{attribute 'c++_compatible'}
FUNCTION_BLOCK JsonSaxHandler_RobotState IMPLEMENTS ITcJsonSaxHandler
VAR_INPUT
END_VAR
VAR_OUTPUT
	parsedState :	STRING;
END_VAR
VAR
	bStateFound :			BOOL := FALSE;
	bCtrlexecstateFound :	BOOL := FALSE;
END_VAR

(* Example JSON

	{
		"_links": {
			"base": {
				"href": "http://127.0.0.1:80/rw/rapid/"
			},
			"self": {
				"href": "execution"
			}
		},
		"status": {
			"code": 294912
		},
		"state": [
			{
				"_type": "rap-execution",
				"_title": "execution",
				"ctrlexecstate": "stopped",
				"cycle": "forever"
			}
		]
	}

*)

{attribute 'TcTypeSystem'}
{attribute 'no-analysis'}
{attribute 'c++_compatible'}
{attribute 'minimal_input_size' := '4'}
{attribute 'pack_mode' := '4'}
{warning 'add method implementation '}
METHOD OnBool : HRESULT
VAR_INPUT
	value	: BOOL;
END_VAR
END_METHOD

{attribute 'TcTypeSystem'}
{attribute 'no-analysis'}
{attribute 'c++_compatible'}
{attribute 'minimal_input_size' := '4'}
{attribute 'pack_mode' := '4'}
{warning 'add method implementation '}
METHOD OnDint : HRESULT
VAR_INPUT
	value	: DINT;
END_VAR
END_METHOD

{attribute 'TcTypeSystem'}
{attribute 'no-analysis'}
{attribute 'c++_compatible'}
{attribute 'minimal_input_size' := '4'}
{attribute 'pack_mode' := '4'}
{warning 'add method implementation '}
METHOD OnEndArray : HRESULT
VAR_INPUT
	elementCount	: UDINT;
END_VAR
END_METHOD

{attribute 'TcTypeSystem'}
{attribute 'no-analysis'}
{attribute 'c++_compatible'}
{attribute 'minimal_input_size' := '4'}
{attribute 'pack_mode' := '4'}
{warning 'add method implementation '}
METHOD OnEndObject : HRESULT
VAR_INPUT
	memberCount	: UDINT;
END_VAR
END_METHOD

{attribute 'TcTypeSystem'}
{attribute 'no-analysis'}
{attribute 'c++_compatible'}
{attribute 'minimal_input_size' := '4'}
{attribute 'pack_mode' := '4'}
{warning 'add method implementation '}
METHOD OnKey : HRESULT
VAR_IN_OUT CONSTANT
	key	: STRING;
END_VAR
VAR_INPUT
	len	: UDINT;
END_VAR


IF (key = 'state') THEN
	bStateFound := TRUE;
END_IF

IF bStateFound AND (key = 'ctrlexecstate') THEN
	bCtrlexecstateFound := TRUE;
END_IF
END_METHOD

{attribute 'TcTypeSystem'}
{attribute 'no-analysis'}
{attribute 'c++_compatible'}
{attribute 'minimal_input_size' := '4'}
{attribute 'pack_mode' := '4'}
{warning 'add method implementation '}
METHOD OnLint : HRESULT
VAR_INPUT
	value	: LINT;
END_VAR
END_METHOD

{attribute 'TcTypeSystem'}
{attribute 'no-analysis'}
{attribute 'c++_compatible'}
{attribute 'minimal_input_size' := '4'}
{attribute 'pack_mode' := '4'}
{warning 'add method implementation '}
METHOD OnLreal : HRESULT
VAR_INPUT
	value	: LREAL;
END_VAR
END_METHOD

{attribute 'TcTypeSystem'}
{attribute 'no-analysis'}
{attribute 'c++_compatible'}
{attribute 'minimal_input_size' := '4'}
{attribute 'pack_mode' := '4'}
{warning 'add method implementation '}
METHOD OnNull : HRESULT
END_METHOD

{attribute 'TcTypeSystem'}
{attribute 'no-analysis'}
{attribute 'c++_compatible'}
{attribute 'minimal_input_size' := '4'}
{attribute 'pack_mode' := '4'}
{warning 'add method implementation '}
METHOD OnRawNumber : HRESULT
VAR_IN_OUT CONSTANT
	value	: STRING;
END_VAR
VAR_INPUT
	len	: UDINT;
END_VAR
END_METHOD

{attribute 'TcTypeSystem'}
{attribute 'no-analysis'}
{attribute 'c++_compatible'}
{attribute 'minimal_input_size' := '4'}
{attribute 'pack_mode' := '4'}
{warning 'add method implementation '}
METHOD OnStartArray : HRESULT
END_METHOD

{attribute 'TcTypeSystem'}
{attribute 'no-analysis'}
{attribute 'c++_compatible'}
{attribute 'minimal_input_size' := '4'}
{attribute 'pack_mode' := '4'}
{warning 'add method implementation '}
METHOD OnStartObject : HRESULT
END_METHOD

{attribute 'TcTypeSystem'}
{attribute 'no-analysis'}
{attribute 'c++_compatible'}
{attribute 'minimal_input_size' := '4'}
{attribute 'pack_mode' := '4'}
{warning 'add method implementation '}
METHOD OnString : HRESULT
VAR_IN_OUT CONSTANT
	value	: STRING;
END_VAR
VAR_INPUT
	len	: UDINT;
END_VAR

IF bCtrlexecstateFound THEN
	parsedState := value;
	OnString := S_FALSE;
END_IF
END_METHOD

{attribute 'TcTypeSystem'}
{attribute 'no-analysis'}
{attribute 'c++_compatible'}
{attribute 'minimal_input_size' := '4'}
{attribute 'pack_mode' := '4'}
{warning 'add method implementation '}
METHOD OnUdint : HRESULT
VAR_INPUT
	value	: UDINT;
END_VAR
END_METHOD

{attribute 'TcTypeSystem'}
{attribute 'no-analysis'}
{attribute 'c++_compatible'}
{attribute 'minimal_input_size' := '4'}
{attribute 'pack_mode' := '4'}
{warning 'add method implementation '}
METHOD OnUlint : HRESULT
VAR_INPUT
	value	: ULINT;
END_VAR
END_METHOD

METHOD Reset : bool
VAR_INPUT
END_VAR

VAR
	bStateFound: BOOL;
END_VAR

// Reset parsing state variables
bStateFound := FALSE;
bCtrlexecstateFound := FALSE;
END_METHOD

{attribute 'TcTypeSystem'}
{attribute 'no-analysis'}
{attribute 'c++_compatible'}
{attribute 'minimal_input_size' := '4'}
{attribute 'pack_mode' := '4'}
{warning 'add method implementation '}
METHOD TcAddRef : UDINT
END_METHOD

{attribute 'TcTypeSystem'}
{attribute 'no-analysis'}
{attribute 'c++_compatible'}
{attribute 'minimal_input_size' := '4'}
{attribute 'pack_mode' := '4'}
{warning 'add method implementation '}
METHOD TcQueryInterface : HRESULT
VAR_INPUT
	iid	: REFERENCE TO IID;
	pipItf	: POINTER TO PVOID;
END_VAR
END_METHOD

{attribute 'TcTypeSystem'}
{attribute 'no-analysis'}
{attribute 'c++_compatible'}
{attribute 'minimal_input_size' := '4'}
{attribute 'pack_mode' := '4'}
{warning 'add method implementation '}
METHOD TcRelease : UDINT
END_METHOD

END_FUNCTION_BLOCK

(* stored: Version 1.1.0.1, ProductVersion 3.1.4024.12
   POU JsonSaxHandler_RobotState: Id {b78b5962-e88f-45fd-9428-34c0448eb750}, SpecialFunc None
   Method OnBool: Id {a8bc2ecd-7eea-4493-a462-cbe13f3242fd}
   Method OnDint: Id {29d2b2b9-7237-49cd-9084-3f0f44c317b4}
   Method OnEndArray: Id {0391a5fd-ef8a-4caf-b3c9-24c17e026c2a}
   Method OnEndObject: Id {1c08a774-1c52-4db3-a402-0aa746cc3c2c}
   Method OnKey: Id {f813b109-3a0c-4827-a2f7-a3de3156088b}
   Method OnLint: Id {c93d24da-b0b2-4c38-b080-f3f010bd8a4c}
   Method OnLreal: Id {5dd3c13e-a549-4927-a2bf-e51021cc6807}
   Method OnNull: Id {6aae938c-b564-45bb-9aa1-3b1d831fad89}
   Method OnRawNumber: Id {bbd27fb8-e2f1-4f8d-9ed6-a029058dfa29}
   Method OnStartArray: Id {c2ceffd3-80e7-457c-bd9f-48d2498d16ed}
   Method OnStartObject: Id {3e06b366-c040-43ef-9843-76b9254ba07a}
   Method OnString: Id {775efc87-98f5-41ea-b2d5-834b680d064c}
   Method OnUdint: Id {bbfc3497-4c52-4175-8776-407bdae20aa2}
   Method OnUlint: Id {988e5f19-06d5-444c-9895-4347f62e9798}
   Method Reset: Id {3c8030e8-783a-4ded-a526-5965c6a5dd36}
   Method TcAddRef: Id {ab820f5c-6937-48d2-a9ba-1dc25b9d1cd9}
   Method TcQueryInterface: Id {b98f40bd-bfcf-447d-93db-882276487a47}
   Method TcRelease: Id {7364fadc-880c-4502-8676-566369b0d118} *)
